TYPE E_CircuitBreakerFault :
(
    NONE := 0,              // Arıza yok
    SPRING_CHARGE := 1,     // Yay kurma arızası
    FEEDBACK := 2,          // Geri besleme hatası
    MOTION_TIMEOUT := 3,    // Hareket zaman aşımı
    TRIP_COIL := 4,         // Trip bobini arızası
    CONTROL_VOLTAGE := 5    // Kontrol gerilimi arızası
);
END_TYPE

(* stored: Version 1.1.0.1, ProductVersion 3.1.4024.15
   EnumerationTextList E_CircuitBreakerFault: Id {d25b2458-a7f2-4be7-81f1-f0c02e2faccb} *)
